FUNCTION_BLOCK TestComposite
  (* Version 0.1, 2005-06-15, Author Name, Chalmers *)
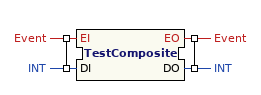
  EVENT_INPUT
    EI WITH DI;
  END_EVENT
  EVENT_OUTPUT
    EO WITH DO;
  END_EVENT
  VAR_INPUT
    DI : INT;
  END_VAR
  VAR_OUTPUT
    DO : INT;
  END_VAR
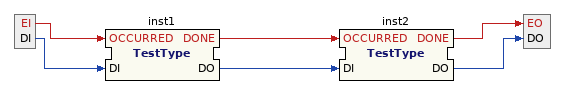
  FBS
    inst1 : TestType;
    inst2 : TestType;
  END_FBS
  EVENT_CONNECTIONS
    EI TO inst1.OCCURRED;
    inst1.DONE TO inst2.OCCURRED;
    inst2.DONE TO EO;
  END_CONNECTIONS
  DATA_CONNECTIONS
    DI TO inst1.DI;
    inst1.DO TO inst2.DI;
    inst2.DO TO DO;
  END_CONNECTIONS
END_FUNCTION_BLOCK
